(* IEC 61131-3 sources: verifaps-lib/share/PPU.stold (part 19) *)

        Stamp_states_t#StampProcess:
            {* begin(State) *}
            {* begin(onEntry) *}
            Stamp$_transit := FALSE;
            {* end(onEntry) *}
            {* begin(onActive) *}
            Stamp$StampSliderMovedIn := FALSE;
            Stamp$StampPusher := TRUE;
            {* end(onActive) *}
            {* begin(transition) *}
            IF Stamp$StampLowered THEN
                Stamp$_transit := TRUE;
                Stamp$_state := Stamp_states_t#Step1;
            END_IF;
            {* end(transition) *}
            {* begin(onExit) *}
            {* end(onExit) *}
            {* end(State) *}

        Stamp_states_t#StampSliderBack:
            {* begin(State) *}
            {* begin(onEntry) *}
            Stamp$_transit := FALSE;
            {* end(onEntry) *}
            {* begin(onActive) *}
            Stamp$StampSliderMovedIn := TRUE;
            Stamp$StampSliderMovedOut := FALSE;
            {* end(onActive) *}
            {* begin(transition) *}
            IF Stamp$StampSliderSensorMovedIn THEN
                Stamp$_transit := TRUE;
                Stamp$_state := Stamp_states_t#StampProcess;
            END_IF;
            {* end(transition) *}
            {* begin(onExit) *}
            {* end(onExit) *}
            {* end(State) *}

        Stamp_states_t#StampSliderForward:
            {* begin(State) *}
            {* begin(onEntry) *}
            Stamp$_transit := FALSE;
            {* end(onEntry) *}
            {* begin(onActive) *}
            Stamp$StampPusher := FALSE;
            Stamp$StampSliderMovedOut := TRUE;
            IF ((Stamp$StampLowered = FALSE) AND (Stamp$StampUp = TRUE)) THEN
                Stamp$interconnect := FALSE;
            END_IF;
            Stamp$Timer$IN := FALSE;
            Stamp$Timer$PT := USINT#0;
            IF Stamp$Timer$IN THEN
                Stamp$Timer$Q := (Stamp$Timer$ET = USINT#0);
                IF (Stamp$Timer$ET > USINT#0) THEN
                    Stamp$Timer$ET := (Stamp$Timer$ET - USINT#1);
                ELSE
                    Stamp$Timer$ET := USINT#0;
                END_IF;
            ELSE
                Stamp$Timer$Q := FALSE;
                Stamp$Timer$ET := Stamp$Timer$PT;
            END_IF;
            {* end(onActive) *}
            {* begin(transition) *}
            IF Stamp$StampSliderMovedOut THEN
                Stamp$_transit := TRUE;
                Stamp$_state := Stamp_states_t#Step2;
            END_IF;
            {* end(transition) *}
            {* begin(onExit) *}
            {* end(onExit) *}
            {* end(State) *}

        Stamp_states_t#Stamp_Init_1:
            {* begin(State) *}
            {* begin(onEntry) *}
            Stamp$_transit := FALSE;
            {* end(onEntry) *}
            {* begin(onActive) *}
            Stamp$StampSliderMovedIn := TRUE;
            Stamp$StampSliderMovedOut := FALSE;
            {* end(onActive) *}
            {* begin(transition) *}
            IF Stamp$StampSliderSensorMovedIn THEN
                Stamp$_transit := TRUE;
                Stamp$_state := Stamp_states_t#Stamp_Init_2;
            END_IF;
            {* end(transition) *}
            {* begin(onExit) *}
            {* end(onExit) *}
            {* end(State) *}

        Stamp_states_t#Stamp_Init_2:
            {* begin(State) *}
            {* begin(onEntry) *}
            Stamp$_transit := FALSE;
            {* end(onEntry) *}
            {* begin(onActive) *}
            Stamp$StampSliderMovedIn := FALSE;
            Stamp$StampSliderMovedOut := TRUE;
            {* end(onActive) *}
            {* begin(transition) *}
            IF Stamp$StampSliderSensorMovedOut THEN
                Stamp$_transit := TRUE;
                Stamp$_state := Stamp_states_t#Stamp_Init_3;
            END_IF;
            {* end(transition) *}
            {* begin(onExit) *}
            {* end(onExit) *}
            {* end(State) *}

        Stamp_states_t#Stamp_Init_3:
            {* begin(State) *}
            {* begin(onEntry) *}
            Stamp$_transit := FALSE;
            {* end(onEntry) *}
            {* begin(onActive) *}
            Stamp$StampPusher := TRUE;
            {* end(onActive) *}
            {* begin(transition) *}
            IF Stamp$StampLowered THEN
                Stamp$_transit := TRUE;
                Stamp$_state := Stamp_states_t#Stamp_Init_4;
            END_IF;
            {* end(transition) *}
            {* begin(onExit) *}
            {* end(onExit) *}
            {* end(State) *}

        Stamp_states_t#Stamp_Init_4:
            {* begin(State) *}
            {* begin(onEntry) *}
            Stamp$_transit := FALSE;
            {* end(onEntry) *}
            {* begin(onActive) *}
            Stamp$StampPusher := FALSE;
            {* end(onActive) *}
            {* begin(transition) *}
            IF Stamp$StampUp THEN
                Stamp$_transit := TRUE;
                Stamp$_state := Stamp_states_t#Interstep;
            END_IF;
            {* end(transition) *}
            {* begin(onExit) *}
            {* end(onExit) *}
            {* end(State) *}

        Stamp_states_t#Start_Stamp:
            {* begin(State) *}
            {* begin(onEntry) *}
            Stamp$_transit := FALSE;
            {* end(onEntry) *}
            {* begin(onActive) *}
            Stamp$StampSliderMovedOut := FALSE;
            Stamp$StampSliderMovedIn := FALSE;
            Stamp$StampPusher := FALSE;
            Stamp$StampGreenLamp := FALSE;
            Stamp$StampPressure := FALSE;
            Stamp$StartCommandStamp := FALSE;
            IF (Stamp$StampStartButton = TRUE) THEN
                Stamp$interconnectStampStartCommand := TRUE;
            END_IF;
            {* end(onActive) *}
            {* begin(transition) *}
            IF Stamp$interconnectStampStartCommand THEN
                Stamp$_transit := TRUE;
                Stamp$_state := Stamp_states_t#Green_Lamp;
            END_IF;
            {* end(transition) *}
            {* begin(onExit) *}
            {* end(onExit) *}
            {* end(State) *}

        Stamp_states_t#Step0:
            {* begin(State) *}
            {* begin(onEntry) *}
            Stamp$_transit := FALSE;
            {* end(onEntry) *}
            {* begin(onActive) *}
            {* end(onActive) *}
            {* begin(transition) *}
            IF Stamp$CraneUp THEN
                Stamp$_transit := TRUE;
                Stamp$_state := Stamp_states_t#StampSliderBack;
            END_IF;
            {* end(transition) *}
            {* begin(onExit) *}
            {* end(onExit) *}
            {* end(State) *}

        Stamp_states_t#Step1:
            {* begin(State) *}
            {* begin(onEntry) *}
            Stamp$_transit := FALSE;
            {* end(onEntry) *}
            {* begin(onActive) *}
            Stamp$Timer$IN := Stamp$StampLowered;
            Stamp$Timer$PT := USINT#0;
            IF Stamp$Timer$IN THEN
                Stamp$Timer$Q := (Stamp$Timer$ET = USINT#0);
                IF (Stamp$Timer$ET > USINT#0) THEN
                    Stamp$Timer$ET := (Stamp$Timer$ET - USINT#1);
                ELSE
                    Stamp$Timer$ET := USINT#0;
                END_IF;
            ELSE
                Stamp$Timer$Q := FALSE;
                Stamp$Timer$ET := Stamp$Timer$PT;
            END_IF;
            Stamp$interconnect := Stamp$Timer$Q;
            {* end(onActive) *}
            {* begin(transition) *}
            IF Stamp$interconnect THEN
                Stamp$_transit := TRUE;
                Stamp$_state := Stamp_states_t#StampSliderForward;
            END_IF;
            {* end(transition) *}
            {* begin(onExit) *}
            {* end(onExit) *}
            {* end(State) *}

        Stamp_states_t#Step2:
            {* begin(State) *}
            {* begin(onEntry) *}
            Stamp$_transit := FALSE;
            {* end(onEntry) *}
            {* begin(onActive) *}
            {* end(onActive) *}
            {* begin(transition) *}
            IF (((Stamp$AnalogCranePosition > INT#16160) AND (Stamp$AnalogCranePosition < INT#16260)) AND NOT Stamp$StampSliderFilled) THEN
                Stamp$_transit := TRUE;
                Stamp$_state := Stamp_states_t#Interstep;
            END_IF;
            {* end(transition) *}
            {* begin(onExit) *}
            {* end(onExit) *}
            {* end(State) *}

            END_CASE;
    CASE Conveyor$_state OF
        Conveyor_states_t#Conveyor_Init:
            {* begin(State) *}
            {* begin(onEntry) *}
            Conveyor$_transit := FALSE;
            {* end(onEntry) *}
            {* begin(onActive) *}
            Conveyor$SorterConveyorTowardsStacker := TRUE;
            Conveyor$SorterConveyorTowardsCrane := FALSE;
            Conveyor$Timer_Conveyor_Test$IN := TRUE;
            Conveyor$Timer_Conveyor_Test$PT := Conveyor$Duration_Conveyor_Test;
            IF Conveyor$Timer_Conveyor_Test$IN THEN
                Conveyor$Timer_Conveyor_Test$Q := (Conveyor$Timer_Conveyor_Test$ET = USINT#0);
                IF (Conveyor$Timer_Conveyor_Test$ET > USINT#0) THEN
                    Conveyor$Timer_Conveyor_Test$ET := (Conveyor$Timer_Conveyor_Test$ET - USINT#1);
                ELSE
                    Conveyor$Timer_Conveyor_Test$ET := USINT#0;
                END_IF;
            ELSE
                Conveyor$Timer_Conveyor_Test$Q := FALSE;
                Conveyor$Timer_Conveyor_Test$ET := Conveyor$Timer_Conveyor_Test$PT;
            END_IF;
            Conveyor$interconnect_Conveyor_Test := Conveyor$Timer_Conveyor_Test$Q;
            {* end(onActive) *}
            {* begin(transition) *}
            IF Conveyor$interconnect_Conveyor_Test THEN
                Conveyor$_transit := TRUE;
                Conveyor$_state := Conveyor_states_t#Conveyor_init_2;
            END_IF;
            {* end(transition) *}
            {* begin(onExit) *}
            {* end(onExit) *}
            {* end(State) *}

        Conveyor_states_t#Conveyor_Stop_Empty_Magazin:
            {* begin(State) *}
            {* begin(onEntry) *}
            Conveyor$_transit := FALSE;
            {* end(onEntry) *}
            {* begin(onActive) *}
            Conveyor$SorterConveyorTowardsStacker := FALSE;
            Conveyor$SorterConveyorTowardsCrane := FALSE;
            Conveyor$interconnectConveyorStartCommand := FALSE;
            {* end(onActive) *}
            {* begin(transition) *}
            IF TRUE THEN
                Conveyor$_transit := TRUE;
                Conveyor$_state := Conveyor_states_t#Interstep;
            END_IF;
            {* end(transition) *}
            {* begin(onExit) *}
            {* end(onExit) *}
            {* end(State) *}

        Conveyor_states_t#Conveyor_Towards_Stacker:
            {* begin(State) *}
            {* begin(onEntry) *}
            Conveyor$_transit := FALSE;
            {* end(onEntry) *}
            {* begin(onActive) *}
            Conveyor$SorterConveyorTowardsStacker := TRUE;
            Conveyor$SorterConveyorTowardsCrane := FALSE;
            {* end(onActive) *}
            {* begin(transition) *}
            IF TRUE THEN
                Conveyor$_transit := TRUE;
                Conveyor$_state := Conveyor_states_t#Runtime_Conveyor;
            END_IF;
            {* end(transition) *}
            {* begin(onExit) *}
            {* end(onExit) *}
            {* end(State) *}

        Conveyor_states_t#Conveyor_init_2:
            {* begin(State) *}
            {* begin(onEntry) *}
            Conveyor$_transit := FALSE;
            {* end(onEntry) *}
            {* begin(onActive) *}
            Conveyor$SorterConveyorTowardsStacker := FALSE;
            Conveyor$SorterConveyorTowardsCrane := FALSE;
            Conveyor$interconnect_Conveyor_Test := FALSE;
            Conveyor$Timer_Conveyor_Test$IN := FALSE;
            Conveyor$Timer_Conveyor_Test$PT := USINT#0;
            IF Conveyor$Timer_Conveyor_Test$IN THEN
                Conveyor$Timer_Conveyor_Test$Q := (Conveyor$Timer_Conveyor_Test$ET = USINT#0);
                IF (Conveyor$Timer_Conveyor_Test$ET > USINT#0) THEN
                    Conveyor$Timer_Conveyor_Test$ET := (Conveyor$Timer_Conveyor_Test$ET - USINT#1);
                ELSE
                    Conveyor$Timer_Conveyor_Test$ET := USINT#0;
                END_IF;
            ELSE
                Conveyor$Timer_Conveyor_Test$Q := FALSE;
                Conveyor$Timer_Conveyor_Test$ET := Conveyor$Timer_Conveyor_Test$PT;
            END_IF;
            {* end(onActive) *}
            {* begin(transition) *}
            IF TRUE THEN
                Conveyor$_transit := TRUE;
                Conveyor$_state := Conveyor_states_t#Interstep;
            END_IF;
            {* end(transition) *}
            {* begin(onExit) *}
            {* end(onExit) *}
            {* end(State) *}

        Conveyor_states_t#Conveyor_pause:
            {* begin(State) *}
            {* begin(onEntry) *}
            Conveyor$_transit := FALSE;
            {* end(onEntry) *}
            {* begin(onActive) *}
            Conveyor$SorterConveyorTowardsStacker := FALSE;
            Conveyor$SorterConveyorTowardsCrane := FALSE;
            Conveyor$interconnect_Conveyor_Runtime := FALSE;
            Conveyor$Timer_Conveyor_Runtime$IN := FALSE;
            Conveyor$Timer_Conveyor_Runtime$PT := USINT#0;
            IF Conveyor$Timer_Conveyor_Runtime$IN THEN
                Conveyor$Timer_Conveyor_Runtime$Q := (Conveyor$Timer_Conveyor_Runtime$ET = USINT#0);
                IF (Conveyor$Timer_Conveyor_Runtime$ET > USINT#0) THEN
                    Conveyor$Timer_Conveyor_Runtime$ET := (Conveyor$Timer_Conveyor_Runtime$ET - USINT#1);
                ELSE
                    Conveyor$Timer_Conveyor_Runtime$ET := USINT#0;
                END_IF;
            ELSE
                Conveyor$Timer_Conveyor_Runtime$Q := FALSE;
                Conveyor$Timer_Conveyor_Runtime$ET := Conveyor$Timer_Conveyor_Runtime$PT;
            END_IF;
            {* end(onActive) *}
            {* begin(transition) *}
            IF TRUE THEN
                Conveyor$_transit := TRUE;
                Conveyor$_state := Conveyor_states_t#Interstep;
            END_IF;
            {* end(transition) *}
            {* begin(onExit) *}
            {* end(onExit) *}
            {* end(State) *}

        Conveyor_states_t#Green_Lamp:
            {* begin(State) *}
            {* begin(onEntry) *}
            Conveyor$_transit := FALSE;
            {* end(onEntry) *}
            {* begin(onActive) *}
            Conveyor$SorterGreenLampConveyor := TRUE;
            Conveyor$interconnectConveyorStartCommand := FALSE;
            {* end(onActive) *}
            {* begin(transition) *}
            IF TRUE THEN
                Conveyor$_transit := TRUE;
                Conveyor$_state := Conveyor_states_t#Conveyor_Init;
            END_IF;
            {* end(transition) *}
            {* begin(onExit) *}
            {* end(onExit) *}
            {* end(State) *}

        Conveyor_states_t#Init:
            {* begin(State) *}
            {* begin(onEntry) *}
            Conveyor$_transit := FALSE;
            {* end(onEntry) *}
            {* begin(onActive) *}
            {* end(onActive) *}
            {* begin(transition) *}
            IF TRUE THEN
                Conveyor$_transit := TRUE;
                Conveyor$_state := Conveyor_states_t#Start_Conveyor;
            END_IF;
            {* end(transition) *}
            {* begin(onExit) *}
            {* end(onExit) *}
            {* end(State) *}

        Conveyor_states_t#Interstep:
            {* begin(State) *}
            {* begin(onEntry) *}
            Conveyor$_transit := FALSE;
            {* end(onEntry) *}
            {* begin(onActive) *}
            Conveyor$StartCommandConveyor := TRUE;
            {* end(onActive) *}
            {* begin(transition) *}
            IF Conveyor$StartVar THEN
                Conveyor$_transit := TRUE;
                Conveyor$_state := Conveyor_states_t#Step0;
            END_IF;
            {* end(transition) *}
            {* begin(onExit) *}
            {* end(onExit) *}
            {* end(State) *}

        Conveyor_states_t#Runtime_Conveyor:
            {* begin(State) *}
            {* begin(onEntry) *}
            Conveyor$_transit := FALSE;
            {* end(onEntry) *}
            {* begin(onActive) *}
            Conveyor$Timer_Conveyor_Runtime$IN := TRUE;
            Conveyor$Timer_Conveyor_Runtime$PT := Conveyor$Duration_Conveyor_Runtime;
            IF Conveyor$Timer_Conveyor_Runtime$IN THEN
                Conveyor$Timer_Conveyor_Runtime$Q := (Conveyor$Timer_Conveyor_Runtime$ET = USINT#0);
                IF (Conveyor$Timer_Conveyor_Runtime$ET > USINT#0) THEN
                    Conveyor$Timer_Conveyor_Runtime$ET := (Conveyor$Timer_Conveyor_Runtime$ET - USINT#1);
                ELSE
                    Conveyor$Timer_Conveyor_Runtime$ET := USINT#0;
                END_IF;
            ELSE
                Conveyor$Timer_Conveyor_Runtime$Q := FALSE;
                Conveyor$Timer_Conveyor_Runtime$ET := Conveyor$Timer_Conveyor_Runtime$PT;
            END_IF;
            Conveyor$interconnect_Conveyor_Runtime := Conveyor$Timer_Conveyor_Runtime$Q;
            {* end(onActive) *}
            {* begin(transition) *}
            IF Conveyor$interconnect_Conveyor_Runtime THEN
                Conveyor$_transit := TRUE;
                Conveyor$_state := Conveyor_states_t#Conveyor_pause;
            END_IF;
            {* end(transition) *}
            {* begin(onExit) *}
            {* end(onExit) *}
            {* end(State) *}

        Conveyor_states_t#Start_Conveyor:
            {* begin(State) *}
            {* begin(onEntry) *}
            Conveyor$_transit := FALSE;
            {* end(onEntry) *}
            {* begin(onActive) *}
            Conveyor$interconnectConveyorTerminationCommand := FALSE;
            Conveyor$SorterConveyorTowardsStacker := FALSE;
            Conveyor$SorterConveyorTowardsCrane := FALSE;
            Conveyor$SorterGreenLampConveyor := FALSE;
            Conveyor$interconnect_Conveyor_Runtime := FALSE;
            Conveyor$interconnect_Conveyor_Test := FALSE;
            Conveyor$Timer_Conveyor_Test$IN := FALSE;
            Conveyor$Timer_Conveyor_Test$PT := USINT#0;
            IF Conveyor$Timer_Conveyor_Test$IN THEN
                Conveyor$Timer_Conveyor_Test$Q := (Conveyor$Timer_Conveyor_Test$ET = USINT#0);
                IF (Conveyor$Timer_Conveyor_Test$ET > USINT#0) THEN
                    Conveyor$Timer_Conveyor_Test$ET := (Conveyor$Timer_Conveyor_Test$ET - USINT#1);
                ELSE
                    Conveyor$Timer_Conveyor_Test$ET := USINT#0;
                END_IF;
            ELSE
                Conveyor$Timer_Conveyor_Test$Q := FALSE;
                Conveyor$Timer_Conveyor_Test$ET := Conveyor$Timer_Conveyor_Test$PT;
            END_IF;
            Conveyor$Timer_Conveyor_Runtime$IN := FALSE;
            Conveyor$Timer_Conveyor_Runtime$PT := USINT#0;
            IF Conveyor$Timer_Conveyor_Runtime$IN THEN
                Conveyor$Timer_Conveyor_Runtime$Q := (Conveyor$Timer_Conveyor_Runtime$ET = USINT#0);
                IF (Conveyor$Timer_Conveyor_Runtime$ET > USINT#0) THEN
                    Conveyor$Timer_Conveyor_Runtime$ET := (Conveyor$Timer_Conveyor_Runtime$ET - USINT#1);
                ELSE
                    Conveyor$Timer_Conveyor_Runtime$ET := USINT#0;
                END_IF;
            ELSE
                Conveyor$Timer_Conveyor_Runtime$Q := FALSE;
                Conveyor$Timer_Conveyor_Runtime$ET := Conveyor$Timer_Conveyor_Runtime$PT;
            END_IF;
            Conveyor$StartVar := FALSE;
            Conveyor$StartCommandConveyor := FALSE;
            IF (Conveyor$SorterStartButton = TRUE) THEN
                Conveyor$interconnectConveyorStartCommand := TRUE;
            END_IF;
            {* end(onActive) *}
            {* begin(transition) *}
            IF Conveyor$interconnectConveyorStartCommand THEN
                Conveyor$_transit := TRUE;
                Conveyor$_state := Conveyor_states_t#Green_Lamp;
            END_IF;
            {* end(transition) *}
            {* begin(onExit) *}
            {* end(onExit) *}
            {* end(State) *}

        Conveyor_states_t#Step0:
            {* begin(State) *}
            {* begin(onEntry) *}
            Conveyor$_transit := FALSE;
            {* end(onEntry) *}
            {* begin(onActive) *}
            {* end(onActive) *}
            {* begin(transition) *}
            IF Conveyor$SorterLightbarrierCraneInterface THEN
                Conveyor$_transit := TRUE;
                Conveyor$_state := Conveyor_states_t#Conveyor_Towards_Stacker;
            ELSEIF NOT Conveyor$SorterLightbarrierCraneInterface THEN
                Conveyor$_transit := TRUE;
                Conveyor$_state := Conveyor_states_t#Conveyor_Stop_Empty_Magazin;
            END_IF;
            {* end(transition) *}
            {* begin(onExit) *}
            {* end(onExit) *}
            {* end(State) *}

            END_CASE;
    CASE Pusher$_state OF
        Pusher_states_t#Check_For_Black:
            {* begin(State) *}
            {* begin(onEntry) *}
            Pusher$_transit := FALSE;
            {* end(onEntry) *}
            {* begin(onActive) *}
            {* end(onActive) *}
            {* begin(transition) *}
            IF ((Pusher$Slide2_black = INT#1) AND (Pusher$Priority_Var_Black = INT#2)) THEN
                Pusher$_transit := TRUE;
                Pusher$_state := Pusher_states_t#Second_Slide_black_workpieces;
            ELSEIF ((Pusher$Slide3_black = INT#1) AND (Pusher$Priority_Var_Black = INT#3)) THEN
                Pusher$_transit := TRUE;
                Pusher$_state := Pusher_states_t#Third_Slide_black_workpieces;
            ELSEIF ((Pusher$Slide1_black = INT#1) AND (Pusher$Priority_Var_Black = INT#1)) THEN
                Pusher$_transit := TRUE;
                Pusher$_state := Pusher_states_t#First_Slide_black_workpieces;
            END_IF;
            {* end(transition) *}
            {* begin(onExit) *}
            {* end(onExit) *}
            {* end(State) *}

        Pusher_states_t#Check_For_Metal:
            {* begin(State) *}
            {* begin(onEntry) *}
            Pusher$_transit := FALSE;
            {* end(onEntry) *}
            {* begin(onActive) *}
            {* end(onActive) *}
            {* begin(transition) *}
            IF ((Pusher$Slide3_metal = INT#1) AND (Pusher$Priority_Var_Metal = INT#3)) THEN
                Pusher$_transit := TRUE;
                Pusher$_state := Pusher_states_t#Third_Slide_metal_workpieces;
            ELSEIF ((Pusher$Slide2_metal = INT#1) AND (Pusher$Priority_Var_Metal = INT#2)) THEN
                Pusher$_transit := TRUE;
                Pusher$_state := Pusher_states_t#Second_Slide_metal_workpieces;
            ELSEIF ((Pusher$Slide1_metal = INT#1) AND (Pusher$Priority_Var_Metal = INT#1)) THEN
                Pusher$_transit := TRUE;
                Pusher$_state := Pusher_states_t#First_Slide_metal_workpieces;
            END_IF;
            {* end(transition) *}
            {* begin(onExit) *}
            {* end(onExit) *}
            {* end(State) *}

        Pusher_states_t#Check_For_White:
            {* begin(State) *}
            {* begin(onEntry) *}
            Pusher$_transit := FALSE;
            {* end(onEntry) *}
            {* begin(onActive) *}
            {* end(onActive) *}
            {* begin(transition) *}
            IF ((Pusher$Slide1_white = INT#1) AND (Pusher$Priority_Var_White = INT#1)) THEN
                Pusher$_transit := TRUE;
                Pusher$_state := Pusher_states_t#First_Slide_white_workpieces;
            ELSEIF ((Pusher$Slide3_white = INT#1) AND (Pusher$Priority_Var_White = INT#3)) THEN
                Pusher$_transit := TRUE;
                Pusher$_state := Pusher_states_t#Third_Slide_white_workpieces;
            ELSEIF ((Pusher$Slide2_white = INT#1) AND (Pusher$Priority_Var_White = INT#2)) THEN
                Pusher$_transit := TRUE;
                Pusher$_state := Pusher_states_t#Second_Slide_white_workpieces;
            END_IF;
            {* end(transition) *}
            {* begin(onExit) *}
            {* end(onExit) *}
            {* end(State) *}

        Pusher_states_t#First_Slide_Timer_Black:
            {* begin(State) *}
            {* begin(onEntry) *}
            Pusher$_transit := FALSE;
            {* end(onEntry) *}
            {* begin(onActive) *}
            IF (Pusher$SorterLightnesssensorCraneInterfaceInverse = TRUE) THEN
                Pusher$Timer_Slide1_Black$IN := Pusher$SorterLightnesssensorCraneInterfaceInverse;
                Pusher$Timer_Slide1_Black$PT := Pusher$Duration_Slide1_Black;
                IF Pusher$Timer_Slide1_Black$IN THEN
                    Pusher$Timer_Slide1_Black$Q := (Pusher$Timer_Slide1_Black$ET = USINT#0);
                    IF (Pusher$Timer_Slide1_Black$ET > USINT#0) THEN
                        Pusher$Timer_Slide1_Black$ET := (Pusher$Timer_Slide1_Black$ET - USINT#1);
                    ELSE
                        Pusher$Timer_Slide1_Black$ET := USINT#0;
                    END_IF;
                ELSE
                    Pusher$Timer_Slide1_Black$Q := FALSE;
                    Pusher$Timer_Slide1_Black$ET := Pusher$Timer_Slide1_Black$PT;
                END_IF;
                Pusher$interconnect_Slide1_Black := Pusher$Timer_Slide1_Black$Q;
            END_IF;
            {* end(onActive) *}
            {* begin(transition) *}
            IF Pusher$interconnect_Slide1_Black THEN
                Pusher$_transit := TRUE;
                Pusher$_state := Pusher_states_t#PusherY1_Move_Out_Black;
            END_IF;
            {* end(transition) *}
            {* begin(onExit) *}
            {* end(onExit) *}
            {* end(State) *}

        Pusher_states_t#First_Slide_Timer_Metal:
            {* begin(State) *}
            {* begin(onEntry) *}
            Pusher$_transit := FALSE;
            {* end(onEntry) *}
            {* begin(onActive) *}
            Pusher$Timer_Slide1_Metal$IN := TRUE;
            Pusher$Timer_Slide1_Metal$PT := Pusher$Duration_Slide1_Metal;
            IF Pusher$Timer_Slide1_Metal$IN THEN
                Pusher$Timer_Slide1_Metal$Q := (Pusher$Timer_Slide1_Metal$ET = USINT#0);
                IF (Pusher$Timer_Slide1_Metal$ET > USINT#0) THEN
                    Pusher$Timer_Slide1_Metal$ET := (Pusher$Timer_Slide1_Metal$ET - USINT#1);
                ELSE
                    Pusher$Timer_Slide1_Metal$ET := USINT#0;
                END_IF;
            ELSE
                Pusher$Timer_Slide1_Metal$Q := FALSE;
                Pusher$Timer_Slide1_Metal$ET := Pusher$Timer_Slide1_Metal$PT;
            END_IF;
            Pusher$interconnect_Slide1_Metal := Pusher$Timer_Slide1_Metal$Q;
            {* end(onActive) *}
            {* begin(transition) *}
            IF Pusher$interconnect_Slide1_Metal THEN
                Pusher$_transit := TRUE;
                Pusher$_state := Pusher_states_t#PusherY1_Move_Out_Metal;
            END_IF;
            {* end(transition) *}
            {* begin(onExit) *}
            {* end(onExit) *}
            {* end(State) *}

        Pusher_states_t#First_Slide_Timer_White:
            {* begin(State) *}
            {* begin(onEntry) *}
            Pusher$_transit := FALSE;
            {* end(onEntry) *}
            {* begin(onActive) *}
            Pusher$Timer_Slide1_White$IN := TRUE;
            Pusher$Timer_Slide1_White$PT := Pusher$Duration_Slide1_White;
            IF Pusher$Timer_Slide1_White$IN THEN
                Pusher$Timer_Slide1_White$Q := (Pusher$Timer_Slide1_White$ET = USINT#0);
                IF (Pusher$Timer_Slide1_White$ET > USINT#0) THEN
                    Pusher$Timer_Slide1_White$ET := (Pusher$Timer_Slide1_White$ET - USINT#1);
                ELSE
                    Pusher$Timer_Slide1_White$ET := USINT#0;
                END_IF;
            ELSE
                Pusher$Timer_Slide1_White$Q := FALSE;
                Pusher$Timer_Slide1_White$ET := Pusher$Timer_Slide1_White$PT;
            END_IF;
            Pusher$interconnect_Slide1_White := Pusher$Timer_Slide1_White$Q;
            {* end(onActive) *}
            {* begin(transition) *}
            IF Pusher$interconnect_Slide1_White THEN
                Pusher$_transit := TRUE;
                Pusher$_state := Pusher_states_t#PusherY1_Move_Out_White;
            END_IF;
            {* end(transition) *}
            {* begin(onExit) *}
            {* end(onExit) *}
            {* end(State) *}

        Pusher_states_t#First_Slide_black_workpieces:
            {* begin(State) *}
            {* begin(onEntry) *}
            Pusher$_transit := FALSE;
            {* end(onEntry) *}
            {* begin(onActive) *}
            {* end(onActive) *}
            {* begin(transition) *}
            IF TRUE THEN
                Pusher$_transit := TRUE;
                Pusher$_state := Pusher_states_t#First_Slide_Timer_Black;
            END_IF;
            {* end(transition) *}
            {* begin(onExit) *}
            {* end(onExit) *}
            {* end(State) *}

        Pusher_states_t#First_Slide_metal_workpieces:
            {* begin(State) *}
            {* begin(onEntry) *}
            Pusher$_transit := FALSE;
            {* end(onEntry) *}
            {* begin(onActive) *}
            {* end(onActive) *}
            {* begin(transition) *}
            IF TRUE THEN
                Pusher$_transit := TRUE;
                Pusher$_state := Pusher_states_t#First_Slide_Timer_Metal;
            END_IF;
            {* end(transition) *}
            {* begin(onExit) *}
            {* end(onExit) *}
            {* end(State) *}

        Pusher_states_t#First_Slide_white_workpieces:
            {* begin(State) *}
            {* begin(onEntry) *}
            Pusher$_transit := FALSE;
            {* end(onEntry) *}
            {* begin(onActive) *}
            {* end(onActive) *}
            {* begin(transition) *}
            IF TRUE THEN
                Pusher$_transit := TRUE;
                Pusher$_state := Pusher_states_t#First_Slide_Timer_White;
            END_IF;
            {* end(transition) *}
            {* begin(onExit) *}
            {* end(onExit) *}
            {* end(State) *}

        Pusher_states_t#Init:
            {* begin(State) *}
            {* begin(onEntry) *}
            Pusher$_transit := FALSE;
            {* end(onEntry) *}
            {* begin(onActive) *}
            {* end(onActive) *}
            {* begin(transition) *}
            IF Pusher$StartVar THEN
                Pusher$_transit := TRUE;
                Pusher$_state := Pusher_states_t#Interstep;
            END_IF;
            {* end(transition) *}
            {* begin(onExit) *}
            {* end(onExit) *}
            {* end(State) *}

        Pusher_states_t#Interstep:
            {* begin(State) *}
            {* begin(onEntry) *}
            Pusher$_transit := FALSE;
            {* end(onEntry) *}
            {* begin(onActive) *}
            Pusher$PusherY1 := FALSE;
            Pusher$PusherY2 := FALSE;
            Pusher$interconnect2 := FALSE;
            Pusher$interconnect3 := FALSE;
            Pusher$StartVar := FALSE;
            Pusher$interconnect_Slide1_Black := FALSE;
            Pusher$interconnect_Slide2_Black := FALSE;
            Pusher$interconnect_Slide1_White := FALSE;
            Pusher$interconnect_Slide2_White := FALSE;
            Pusher$interconnect_Slide1_Metal := FALSE;
            Pusher$interconnect_Slide2_Metal := FALSE;
            {* end(onActive) *}
            {* begin(transition) *}
            IF TRUE THEN
                Pusher$_transit := TRUE;
                Pusher$_state := Pusher_states_t#Interstep_2;
            END_IF;
            {* end(transition) *}
            {* begin(onExit) *}
            {* end(onExit) *}
            {* end(State) *}

        Pusher_states_t#Interstep_2:
            {* begin(State) *}
            {* begin(onEntry) *}
            Pusher$_transit := FALSE;
            {* end(onEntry) *}
            {* begin(onActive) *}
            {* end(onActive) *}
            {* begin(transition) *}
            IF ((Pusher$SorterLightnessSensorPusher1 AND Pusher$SorterCapacitiveSensorPusher1) AND (Pusher$Priority_Var_Metal > INT#0)) THEN
                Pusher$_transit := TRUE;
                Pusher$_state := Pusher_states_t#Check_For_Metal;
            ELSEIF ((NOT Pusher$SorterLightnesssensorCraneInterfaceInverse AND Pusher$SorterLightbarrierCraneInterface) AND (Pusher$Priority_Var_Black > INT#0)) THEN
                Pusher$_transit := TRUE;
                Pusher$_state := Pusher_states_t#Check_For_Black;
            ELSEIF ((Pusher$SorterLightnessSensorPusher1 AND NOT Pusher$SorterCapacitiveSensorPusher1) AND (Pusher$Priority_Var_White > INT#0)) THEN
                Pusher$_transit := TRUE;
                Pusher$_state := Pusher_states_t#Check_For_White;
            END_IF;
            {* end(transition) *}
            {* begin(onExit) *}
            {* end(onExit) *}
            {* end(State) *}

        Pusher_states_t#PusherY1_Move_In_Black:
            {* begin(State) *}
            {* begin(onEntry) *}
            Pusher$_transit := FALSE;
            {* end(onEntry) *}
            {* begin(onActive) *}
            IF ((Pusher$SorterPusher1MovedOut = TRUE) AND (Pusher$SorterPusher1MovedIn = FALSE)) THEN
                Pusher$PusherY1 := FALSE;
            END_IF;
            {* end(onActive) *}
            {* begin(transition) *}
            IF Pusher$SorterPusher1MovedIn THEN
                Pusher$_transit := TRUE;
                Pusher$_state := Pusher_states_t#Reset_interconnect_Slide1_Black;
            END_IF;
            {* end(transition) *}
            {* begin(onExit) *}
            {* end(onExit) *}
            {* end(State) *}

        Pusher_states_t#PusherY1_Move_In_Metal:
            {* begin(State) *}
            {* begin(onEntry) *}
            Pusher$_transit := FALSE;
            {* end(onEntry) *}
            {* begin(onActive) *}
            IF ((Pusher$SorterPusher1MovedOut = TRUE) AND (Pusher$SorterPusher1MovedIn = FALSE)) THEN
                Pusher$PusherY1 := FALSE;
            END_IF;
            {* end(onActive) *}
            {* begin(transition) *}
            IF Pusher$SorterPusher1MovedIn THEN
                Pusher$_transit := TRUE;
                Pusher$_state := Pusher_states_t#Reset_interconnect_Slide1_Metal;
            END_IF;
            {* end(transition) *}
            {* begin(onExit) *}
            {* end(onExit) *}
            {* end(State) *}

        Pusher_states_t#PusherY1_Move_In_White:
            {* begin(State) *}
            {* begin(onEntry) *}
            Pusher$_transit := FALSE;
            {* end(onEntry) *}
            {* begin(onActive) *}
            IF ((Pusher$SorterPusher1MovedOut = TRUE) AND (Pusher$SorterPusher1MovedIn = FALSE)) THEN
                Pusher$PusherY1 := FALSE;
            END_IF;
            {* end(onActive) *}
            {* begin(transition) *}
            IF Pusher$SorterPusher1MovedIn THEN
                Pusher$_transit := TRUE;
                Pusher$_state := Pusher_states_t#Reset_interconnect_Slide1_White;
            END_IF;
            {* end(transition) *}
            {* begin(onExit) *}
            {* end(onExit) *}
            {* end(State) *}

        Pusher_states_t#PusherY1_Move_Out_Black:
            {* begin(State) *}
            {* begin(onEntry) *}
            Pusher$_transit := FALSE;
            {* end(onEntry) *}
            {* begin(onActive) *}
            IF ((Pusher$SorterPusher1MovedOut = FALSE) AND (Pusher$SorterPusher1MovedIn = TRUE)) THEN
                Pusher$PusherY1 := TRUE;
            END_IF;
            {* end(onActive) *}
            {* begin(transition) *}
            IF Pusher$SorterPusher1MovedOut THEN
                Pusher$_transit := TRUE;
                Pusher$_state := Pusher_states_t#Wait_Y1_Black;
            END_IF;
            {* end(transition) *}
            {* begin(onExit) *}
            {* end(onExit) *}
            {* end(State) *}

        Pusher_states_t#PusherY1_Move_Out_Metal:
            {* begin(State) *}
            {* begin(onEntry) *}
            Pusher$_transit := FALSE;
            {* end(onEntry) *}
            {* begin(onActive) *}
            IF ((Pusher$SorterPusher1MovedOut = FALSE) AND (Pusher$SorterPusher1MovedIn = TRUE)) THEN
                Pusher$PusherY1 := TRUE;
            END_IF;
            {* end(onActive) *}
            {* begin(transition) *}
            IF Pusher$SorterPusher1MovedOut THEN
                Pusher$_transit := TRUE;
                Pusher$_state := Pusher_states_t#Wait_Y1_Metal;
            END_IF;
            {* end(transition) *}
            {* begin(onExit) *}
            {* end(onExit) *}
            {* end(State) *}

        Pusher_states_t#PusherY1_Move_Out_White:
            {* begin(State) *}
            {* begin(onEntry) *}
            Pusher$_transit := FALSE;
            {* end(onEntry) *}
            {* begin(onActive) *}
            IF ((Pusher$SorterPusher1MovedOut = FALSE) AND (Pusher$SorterPusher1MovedIn = TRUE)) THEN
                Pusher$PusherY1 := TRUE;
            END_IF;
            {* end(onActive) *}
            {* begin(transition) *}
            IF Pusher$SorterPusher1MovedOut THEN
                Pusher$_transit := TRUE;
                Pusher$_state := Pusher_states_t#Wait_Y1_White;
            END_IF;
            {* end(transition) *}
            {* begin(onExit) *}
            {* end(onExit) *}
            {* end(State) *}

        Pusher_states_t#PusherY2_Move_In_Black:
            {* begin(State) *}
            {* begin(onEntry) *}
            Pusher$_transit := FALSE;
            {* end(onEntry) *}
            {* begin(onActive) *}
            IF ((Pusher$SorterPusher2MovedOut = TRUE) AND (Pusher$SorterPusher2MovedIn = FALSE)) THEN
                Pusher$PusherY2 := FALSE;
            END_IF;
            {* end(onActive) *}
            {* begin(transition) *}
            IF Pusher$SorterPusher2MovedIn THEN
                Pusher$_transit := TRUE;
                Pusher$_state := Pusher_states_t#Reset_interconnect_Slide2_Black;
            END_IF;
            {* end(transition) *}
            {* begin(onExit) *}
            {* end(onExit) *}
            {* end(State) *}

        Pusher_states_t#PusherY2_Move_In_Metal:
            {* begin(State) *}
            {* begin(onEntry) *}
            Pusher$_transit := FALSE;
            {* end(onEntry) *}
            {* begin(onActive) *}
            IF ((Pusher$SorterPusher2MovedOut = TRUE) AND (Pusher$SorterPusher2MovedIn = FALSE)) THEN
                Pusher$PusherY2 := FALSE;
            END_IF;
            {* end(onActive) *}
            {* begin(transition) *}
            IF Pusher$SorterPusher2MovedIn THEN
                Pusher$_transit := TRUE;
                Pusher$_state := Pusher_states_t#Reset_interconnect_Slide2_Metal;
            END_IF;
            {* end(transition) *}
            {* begin(onExit) *}
            {* end(onExit) *}
            {* end(State) *}

        Pusher_states_t#PusherY2_Move_In_White:
            {* begin(State) *}
            {* begin(onEntry) *}
            Pusher$_transit := FALSE;
            {* end(onEntry) *}
            {* begin(onActive) *}
            IF ((Pusher$SorterPusher2MovedOut = TRUE) AND (Pusher$SorterPusher2MovedIn = FALSE)) THEN
                Pusher$PusherY2 := FALSE;
            END_IF;
            {* end(onActive) *}
            {* begin(transition) *}
            IF Pusher$SorterPusher2MovedIn THEN
                Pusher$_transit := TRUE;
                Pusher$_state := Pusher_states_t#Reset_interconnect_Slide2_White;
            END_IF;
            {* end(transition) *}
            {* begin(onExit) *}
            {* end(onExit) *}
            {* end(State) *}

        Pusher_states_t#PusherY2_Move_Out_Black:
            {* begin(State) *}
            {* begin(onEntry) *}
            Pusher$_transit := FALSE;
            {* end(onEntry) *}
            {* begin(onActive) *}
            IF ((Pusher$SorterPusher2MovedOut = FALSE) AND (Pusher$SorterPusher2MovedIn = TRUE)) THEN
                Pusher$PusherY2 := TRUE;
            END_IF;
            {* end(onActive) *}
            {* begin(transition) *}
            IF Pusher$SorterPusher2MovedOut THEN
                Pusher$_transit := TRUE;
                Pusher$_state := Pusher_states_t#Wait_Y2_Black;
            END_IF;
            {* end(transition) *}
            {* begin(onExit) *}
            {* end(onExit) *}
            {* end(State) *}

        Pusher_states_t#PusherY2_Move_Out_Metal:
            {* begin(State) *}
            {* begin(onEntry) *}
            Pusher$_transit := FALSE;
            {* end(onEntry) *}
            {* begin(onActive) *}
            IF ((Pusher$SorterPusher2MovedOut = FALSE) AND (Pusher$SorterPusher2MovedIn = TRUE)) THEN
                Pusher$PusherY2 := TRUE;
            END_IF;
            {* end(onActive) *}
            {* begin(transition) *}
            IF Pusher$SorterPusher2MovedOut THEN
                Pusher$_transit := TRUE;
                Pusher$_state := Pusher_states_t#Wait_Y2_Metal;
            END_IF;
            {* end(transition) *}
            {* begin(onExit) *}
            {* end(onExit) *}
            {* end(State) *}

        Pusher_states_t#PusherY2_Move_Out_White:
            {* begin(State) *}
            {* begin(onEntry) *}
            Pusher$_transit := FALSE;
            {* end(onEntry) *}
            {* begin(onActive) *}
            IF ((Pusher$SorterPusher2MovedOut = FALSE) AND (Pusher$SorterPusher2MovedIn = TRUE)) THEN
                Pusher$PusherY2 := TRUE;
            END_IF;
            {* end(onActive) *}
            {* begin(transition) *}
            IF Pusher$SorterPusher2MovedOut THEN
                Pusher$_transit := TRUE;
                Pusher$_state := Pusher_states_t#Wait_Y2_White;
            END_IF;
            {* end(transition) *}
            {* begin(onExit) *}
            {* end(onExit) *}
            {* end(State) *}

        Pusher_states_t#Reset_interconnect3:
            {* begin(State) *}
            {* begin(onEntry) *}
            Pusher$_transit := FALSE;
            {* end(onEntry) *}
            {* begin(onActive) *}
            Pusher$interconnect2 := FALSE;
            Pusher$Timer2$IN := FALSE;
            Pusher$Timer2$PT := USINT#0;
            IF Pusher$Timer2$IN THEN
                Pusher$Timer2$Q := (Pusher$Timer2$ET = USINT#0);
                IF (Pusher$Timer2$ET > USINT#0) THEN
                    Pusher$Timer2$ET := (Pusher$Timer2$ET - USINT#1);
                ELSE
                    Pusher$Timer2$ET := USINT#0;
                END_IF;
            ELSE
                Pusher$Timer2$Q := FALSE;
                Pusher$Timer2$ET := Pusher$Timer2$PT;
            END_IF;
            Pusher$Slide3_black := (Pusher$Slide3_black - INT#1);
            Pusher$Priority_Var_Black := (Pusher$Priority_Var_Black - INT#1);
            {* end(onActive) *}
            {* begin(transition) *}
            IF TRUE THEN
                Pusher$_transit := TRUE;
                Pusher$_state := Pusher_states_t#Interstep_2;
            END_IF;
            {* end(transition) *}
            {* begin(onExit) *}
            {* end(onExit) *}
            {* end(State) *}

        Pusher_states_t#Reset_interconnect_Slide1_Black:
            {* begin(State) *}
            {* begin(onEntry) *}
            Pusher$_transit := FALSE;
            {* end(onEntry) *}
            {* begin(onActive) *}
            Pusher$interconnect3 := FALSE;
            Pusher$Timer3$IN := FALSE;
            Pusher$Timer3$PT := USINT#0;
            IF Pusher$Timer3$IN THEN
                Pusher$Timer3$Q := (Pusher$Timer3$ET = USINT#0);
                IF (Pusher$Timer3$ET > USINT#0) THEN
                    Pusher$Timer3$ET := (Pusher$Timer3$ET - USINT#1);
                ELSE
                    Pusher$Timer3$ET := USINT#0;
                END_IF;
            ELSE
                Pusher$Timer3$Q := FALSE;
                Pusher$Timer3$ET := Pusher$Timer3$PT;
            END_IF;
            Pusher$interconnect_Slide1_Black := FALSE;
            Pusher$Timer_Slide1_Black$IN := FALSE;
            Pusher$Timer_Slide1_Black$PT := USINT#0;
            IF Pusher$Timer_Slide1_Black$IN THEN
                Pusher$Timer_Slide1_Black$Q := (Pusher$Timer_Slide1_Black$ET = USINT#0);
                IF (Pusher$Timer_Slide1_Black$ET > USINT#0) THEN
                    Pusher$Timer_Slide1_Black$ET := (Pusher$Timer_Slide1_Black$ET - USINT#1);
                ELSE
                    Pusher$Timer_Slide1_Black$ET := USINT#0;
                END_IF;
            ELSE
                Pusher$Timer_Slide1_Black$Q := FALSE;
                Pusher$Timer_Slide1_Black$ET := Pusher$Timer_Slide1_Black$PT;
            END_IF;
            Pusher$Slide1_black := (Pusher$Slide1_black - INT#1);
            Pusher$Priority_Var_Black := (Pusher$Priority_Var_Black - INT#1);
            {* end(onActive) *}
            {* begin(transition) *}
            IF TRUE THEN
                Pusher$_transit := TRUE;
                Pusher$_state := Pusher_states_t#Interstep_2;
            END_IF;
            {* end(transition) *}
            {* begin(onExit) *}
            {* end(onExit) *}
            {* end(State) *}

        Pusher_states_t#Reset_interconnect_Slide1_Metal:
            {* begin(State) *}
            {* begin(onEntry) *}
            Pusher$_transit := FALSE;
            {* end(onEntry) *}
            {* begin(onActive) *}
            Pusher$interconnect3 := FALSE;
            Pusher$Timer3$IN := FALSE;
            Pusher$Timer3$PT := USINT#0;
            IF Pusher$Timer3$IN THEN
                Pusher$Timer3$Q := (Pusher$Timer3$ET = USINT#0);
                IF (Pusher$Timer3$ET > USINT#0) THEN
                    Pusher$Timer3$ET := (Pusher$Timer3$ET - USINT#1);
                ELSE
                    Pusher$Timer3$ET := USINT#0;
                END_IF;
            ELSE
                Pusher$Timer3$Q := FALSE;
                Pusher$Timer3$ET := Pusher$Timer3$PT;
            END_IF;
            Pusher$interconnect_Slide1_Metal := FALSE;
            Pusher$Timer_Slide1_Metal$IN := FALSE;
            Pusher$Timer_Slide1_Metal$PT := USINT#0;
            IF Pusher$Timer_Slide1_Metal$IN THEN
                Pusher$Timer_Slide1_Metal$Q := (Pusher$Timer_Slide1_Metal$ET = USINT#0);
                IF (Pusher$Timer_Slide1_Metal$ET > USINT#0) THEN
                    Pusher$Timer_Slide1_Metal$ET := (Pusher$Timer_Slide1_Metal$ET - USINT#1);
                ELSE
                    Pusher$Timer_Slide1_Metal$ET := USINT#0;
                END_IF;
            ELSE
                Pusher$Timer_Slide1_Metal$Q := FALSE;
                Pusher$Timer_Slide1_Metal$ET := Pusher$Timer_Slide1_Metal$PT;
            END_IF;
            Pusher$Slide1_metal := (Pusher$Slide1_metal - INT#1);
            Pusher$Priority_Var_Metal := (Pusher$Priority_Var_Metal - INT#1);
            {* end(onActive) *}
            {* begin(transition) *}
            IF TRUE THEN
                Pusher$_transit := TRUE;
                Pusher$_state := Pusher_states_t#Interstep_2;
            END_IF;
            {* end(transition) *}
            {* begin(onExit) *}
            {* end(onExit) *}
            {* end(State) *}

        Pusher_states_t#Reset_interconnect_Slide1_White:
            {* begin(State) *}
            {* begin(onEntry) *}
            Pusher$_transit := FALSE;
            {* end(onEntry) *}
            {* begin(onActive) *}
            Pusher$interconnect3 := FALSE;
            Pusher$Timer3$IN := FALSE;
            Pusher$Timer3$PT := USINT#0;
            IF Pusher$Timer3$IN THEN
                Pusher$Timer3$Q := (Pusher$Timer3$ET = USINT#0);
                IF (Pusher$Timer3$ET > USINT#0) THEN
                    Pusher$Timer3$ET := (Pusher$Timer3$ET - USINT#1);
                ELSE
                    Pusher$Timer3$ET := USINT#0;
                END_IF;
            ELSE
                Pusher$Timer3$Q := FALSE;
                Pusher$Timer3$ET := Pusher$Timer3$PT;
            END_IF;
            Pusher$interconnect_Slide1_White := FALSE;
            Pusher$Timer_Slide1_White$IN := FALSE;
            Pusher$Timer_Slide1_White$PT := USINT#0;
            IF Pusher$Timer_Slide1_White$IN THEN
                Pusher$Timer_Slide1_White$Q := (Pusher$Timer_Slide1_White$ET = USINT#0);
                IF (Pusher$Timer_Slide1_White$ET > USINT#0) THEN
                    Pusher$Timer_Slide1_White$ET := (Pusher$Timer_Slide1_White$ET - USINT#1);
                ELSE
                    Pusher$Timer_Slide1_White$ET := USINT#0;
                END_IF;
            ELSE
                Pusher$Timer_Slide1_White$Q := FALSE;
                Pusher$Timer_Slide1_White$ET := Pusher$Timer_Slide1_White$PT;
            END_IF;
            Pusher$Slide1_white := (Pusher$Slide1_white - INT#1);
            Pusher$Priority_Var_White := (Pusher$Priority_Var_White - INT#1);
            {* end(onActive) *}
            {* begin(transition) *}
            IF TRUE THEN
                Pusher$_transit := TRUE;
                Pusher$_state := Pusher_states_t#Interstep_2;
            END_IF;
            {* end(transition) *}
            {* begin(onExit) *}
            {* end(onExit) *}
            {* end(State) *}

        Pusher_states_t#Reset_interconnect_Slide2_Black:
            {* begin(State) *}
            {* begin(onEntry) *}
            Pusher$_transit := FALSE;
            {* end(onEntry) *}
            {* begin(onActive) *}
            Pusher$interconnect3 := FALSE;
            Pusher$Timer3$IN := FALSE;
            Pusher$Timer3$PT := USINT#0;
            IF Pusher$Timer3$IN THEN
                Pusher$Timer3$Q := (Pusher$Timer3$ET = USINT#0);
                IF (Pusher$Timer3$ET > USINT#0) THEN
                    Pusher$Timer3$ET := (Pusher$Timer3$ET - USINT#1);
                ELSE
                    Pusher$Timer3$ET := USINT#0;
                END_IF;
            ELSE
                Pusher$Timer3$Q := FALSE;
                Pusher$Timer3$ET := Pusher$Timer3$PT;
            END_IF;
            Pusher$interconnect_Slide2_Black := FALSE;
            Pusher$Timer_Slide2_Black$IN := FALSE;
            Pusher$Timer_Slide2_Black$PT := USINT#0;
            IF Pusher$Timer_Slide2_Black$IN THEN
                Pusher$Timer_Slide2_Black$Q := (Pusher$Timer_Slide2_Black$ET = USINT#0);
                IF (Pusher$Timer_Slide2_Black$ET > USINT#0) THEN
                    Pusher$Timer_Slide2_Black$ET := (Pusher$Timer_Slide2_Black$ET - USINT#1);
                ELSE
                    Pusher$Timer_Slide2_Black$ET := USINT#0;
                END_IF;
            ELSE
                Pusher$Timer_Slide2_Black$Q := FALSE;
                Pusher$Timer_Slide2_Black$ET := Pusher$Timer_Slide2_Black$PT;
            END_IF;
            Pusher$Slide2_black := (Pusher$Slide2_black - INT#1);
            Pusher$Priority_Var_Black := (Pusher$Priority_Var_Black - INT#1);
            {* end(onActive) *}
            {* begin(transition) *}
            IF TRUE THEN
                Pusher$_transit := TRUE;
                Pusher$_state := Pusher_states_t#Interstep_2;
            END_IF;
            {* end(transition) *}
            {* begin(onExit) *}
            {* end(onExit) *}
            {* end(State) *}

        Pusher_states_t#Reset_interconnect_Slide2_Metal:
            {* begin(State) *}
            {* begin(onEntry) *}
            Pusher$_transit := FALSE;
            {* end(onEntry) *}
            {* begin(onActive) *}
            Pusher$interconnect3 := FALSE;
            Pusher$Timer3$IN := FALSE;
            Pusher$Timer3$PT := USINT#0;
            IF Pusher$Timer3$IN THEN
                Pusher$Timer3$Q := (Pusher$Timer3$ET = USINT#0);
                IF (Pusher$Timer3$ET > USINT#0) THEN
                    Pusher$Timer3$ET := (Pusher$Timer3$ET - USINT#1);
                ELSE
                    Pusher$Timer3$ET := USINT#0;
                END_IF;
            ELSE
                Pusher$Timer3$Q := FALSE;
                Pusher$Timer3$ET := Pusher$Timer3$PT;
            END_IF;
            Pusher$interconnect_Slide2_Metal := FALSE;
            Pusher$Timer_Slide2_Metal$IN := FALSE;
            Pusher$Timer_Slide2_Metal$PT := USINT#0;
            IF Pusher$Timer_Slide2_Metal$IN THEN
                Pusher$Timer_Slide2_Metal$Q := (Pusher$Timer_Slide2_Metal$ET = USINT#0);
                IF (Pusher$Timer_Slide2_Metal$ET > USINT#0) THEN
                    Pusher$Timer_Slide2_Metal$ET := (Pusher$Timer_Slide2_Metal$ET - USINT#1);
                ELSE
                    Pusher$Timer_Slide2_Metal$ET := USINT#0;
                END_IF;
            ELSE
                Pusher$Timer_Slide2_Metal$Q := FALSE;
                Pusher$Timer_Slide2_Metal$ET := Pusher$Timer_Slide2_Metal$PT;
            END_IF;
            Pusher$Slide2_metal := (Pusher$Slide2_metal - INT#1);
            Pusher$Priority_Var_Metal := (Pusher$Priority_Var_Metal - INT#1);
            {* end(onActive) *}
            {* begin(transition) *}
            IF TRUE THEN
                Pusher$_transit := TRUE;
                Pusher$_state := Pusher_states_t#Interstep_2;
            END_IF;
            {* end(transition) *}
            {* begin(onExit) *}
            {* end(onExit) *}
            {* end(State) *}

        Pusher_states_t#Reset_interconnect_Slide2_White:
            {* begin(State) *}
            {* begin(onEntry) *}
            Pusher$_transit := FALSE;
            {* end(onEntry) *}
            {* begin(onActive) *}
            Pusher$interconnect3 := FALSE;
            Pusher$Timer3$IN := FALSE;
            Pusher$Timer3$PT := USINT#0;
            IF Pusher$Timer3$IN THEN
                Pusher$Timer3$Q := (Pusher$Timer3$ET = USINT#0);
                IF (Pusher$Timer3$ET > USINT#0) THEN
                    Pusher$Timer3$ET := (Pusher$Timer3$ET - USINT#1);
                ELSE
                    Pusher$Timer3$ET := USINT#0;
                END_IF;
            ELSE
                Pusher$Timer3$Q := FALSE;
                Pusher$Timer3$ET := Pusher$Timer3$PT;
            END_IF;
            Pusher$interconnect_Slide2_White := FALSE;
            Pusher$Timer_Slide2_White$IN := FALSE;
            Pusher$Timer_Slide2_White$PT := USINT#0;
            IF Pusher$Timer_Slide2_White$IN THEN
                Pusher$Timer_Slide2_White$Q := (Pusher$Timer_Slide2_White$ET = USINT#0);
                IF (Pusher$Timer_Slide2_White$ET > USINT#0) THEN
                    Pusher$Timer_Slide2_White$ET := (Pusher$Timer_Slide2_White$ET - USINT#1);
                ELSE
                    Pusher$Timer_Slide2_White$ET := USINT#0;
                END_IF;
            ELSE
                Pusher$Timer_Slide2_White$Q := FALSE;
                Pusher$Timer_Slide2_White$ET := Pusher$Timer_Slide2_White$PT;
            END_IF;
            Pusher$Slide2_white := (Pusher$Slide2_white - INT#1);
            Pusher$Priority_Var_White := (Pusher$Priority_Var_White - INT#1);
            {* end(onActive) *}
            {* begin(transition) *}
            IF TRUE THEN
                Pusher$_transit := TRUE;
                Pusher$_state := Pusher_states_t#Interstep_2;
            END_IF;
            {* end(transition) *}
            {* begin(onExit) *}
            {* end(onExit) *}
            {* end(State) *}

        Pusher_states_t#Reset_interconnect_Slide3_Metal:
            {* begin(State) *}
            {* begin(onEntry) *}
            Pusher$_transit := FALSE;
            {* end(onEntry) *}
            {* begin(onActive) *}
            Pusher$interconnect3 := FALSE;
            Pusher$Timer3$IN := FALSE;
            Pusher$Timer3$PT := USINT#0;
            IF Pusher$Timer3$IN THEN
                Pusher$Timer3$Q := (Pusher$Timer3$ET = USINT#0);
                IF (Pusher$Timer3$ET > USINT#0) THEN
                    Pusher$Timer3$ET := (Pusher$Timer3$ET - USINT#1);
                ELSE
                    Pusher$Timer3$ET := USINT#0;
                END_IF;
            ELSE
                Pusher$Timer3$Q := FALSE;
                Pusher$Timer3$ET := Pusher$Timer3$PT;
            END_IF;
            Pusher$Slide3_metal := (Pusher$Slide3_metal - INT#1);
            Pusher$Priority_Var_Metal := (Pusher$Priority_Var_Metal - INT#1);
            {* end(onActive) *}
            {* begin(transition) *}
            IF TRUE THEN
                Pusher$_transit := TRUE;
                Pusher$_state := Pusher_states_t#Interstep_2;
            END_IF;
            {* end(transition) *}
            {* begin(onExit) *}
            {* end(onExit) *}
            {* end(State) *}

        Pusher_states_t#Reset_interconnect_Slide3_White:
            {* begin(State) *}
            {* begin(onEntry) *}
            Pusher$_transit := FALSE;
            {* end(onEntry) *}
            {* begin(onActive) *}
            Pusher$interconnect3 := FALSE;
            Pusher$Timer3$IN := FALSE;
            Pusher$Timer3$PT := USINT#0;
            IF Pusher$Timer3$IN THEN
                Pusher$Timer3$Q := (Pusher$Timer3$ET = USINT#0);
                IF (Pusher$Timer3$ET > USINT#0) THEN
                    Pusher$Timer3$ET := (Pusher$Timer3$ET - USINT#1);
                ELSE
                    Pusher$Timer3$ET := USINT#0;
                END_IF;
            ELSE
                Pusher$Timer3$Q := FALSE;
                Pusher$Timer3$ET := Pusher$Timer3$PT;
            END_IF;
            Pusher$Slide3_white := (Pusher$Slide3_white - INT#1);
            Pusher$Priority_Var_White := (Pusher$Priority_Var_White - INT#1);
            {* end(onActive) *}
            {* begin(transition) *}
            IF TRUE THEN
                Pusher$_transit := TRUE;
                Pusher$_state := Pusher_states_t#Interstep_2;
            END_IF;
            {* end(transition) *}
            {* begin(onExit) *}
            {* end(onExit) *}
            {* end(State) *}

        Pusher_states_t#Second_Slide_Timer_Black:
            {* begin(State) *}
            {* begin(onEntry) *}
            Pusher$_transit := FALSE;
            {* end(onEntry) *}
            {* begin(onActive) *}
            IF (Pusher$SorterLightnesssensorCraneInterfaceInverse = TRUE) THEN
                Pusher$Timer_Slide2_Black$IN := Pusher$SorterLightnesssensorCraneInterfaceInverse;
                Pusher$Timer_Slide2_Black$PT := Pusher$Duration_Slide2_Black;
                IF Pusher$Timer_Slide2_Black$IN THEN
                    Pusher$Timer_Slide2_Black$Q := (Pusher$Timer_Slide2_Black$ET = USINT#0);
                    IF (Pusher$Timer_Slide2_Black$ET > USINT#0) THEN
                        Pusher$Timer_Slide2_Black$ET := (Pusher$Timer_Slide2_Black$ET - USINT#1);
                    ELSE
                        Pusher$Timer_Slide2_Black$ET := USINT#0;
                    END_IF;
                ELSE
                    Pusher$Timer_Slide2_Black$Q := FALSE;
                    Pusher$Timer_Slide2_Black$ET := Pusher$Timer_Slide2_Black$PT;
                END_IF;
                Pusher$interconnect_Slide2_Black := Pusher$Timer_Slide2_Black$Q;
            END_IF;
            {* end(onActive) *}
            {* begin(transition) *}
            IF Pusher$interconnect_Slide2_Black THEN
                Pusher$_transit := TRUE;
                Pusher$_state := Pusher_states_t#PusherY2_Move_Out_Black;
            END_IF;
            {* end(transition) *}
            {* begin(onExit) *}
            {* end(onExit) *}
            {* end(State) *}

        Pusher_states_t#Second_Slide_Timer_Metal:
            {* begin(State) *}
            {* begin(onEntry) *}
            Pusher$_transit := FALSE;
            {* end(onEntry) *}
            {* begin(onActive) *}
            Pusher$Timer_Slide2_Metal$IN := TRUE;
            Pusher$Timer_Slide2_Metal$PT := Pusher$Duration_Slide2_Metal;
            IF Pusher$Timer_Slide2_Metal$IN THEN
                Pusher$Timer_Slide2_Metal$Q := (Pusher$Timer_Slide2_Metal$ET = USINT#0);
                IF (Pusher$Timer_Slide2_Metal$ET > USINT#0) THEN
                    Pusher$Timer_Slide2_Metal$ET := (Pusher$Timer_Slide2_Metal$ET - USINT#1);
                ELSE
                    Pusher$Timer_Slide2_Metal$ET := USINT#0;
                END_IF;
            ELSE
                Pusher$Timer_Slide2_Metal$Q := FALSE;
                Pusher$Timer_Slide2_Metal$ET := Pusher$Timer_Slide2_Metal$PT;
            END_IF;
            Pusher$interconnect_Slide2_Metal := Pusher$Timer_Slide2_Metal$Q;
            {* end(onActive) *}
            {* begin(transition) *}
            IF Pusher$interconnect_Slide2_Metal THEN
                Pusher$_transit := TRUE;
                Pusher$_state := Pusher_states_t#PusherY2_Move_Out_Metal;
            END_IF;
            {* end(transition) *}
            {* begin(onExit) *}
            {* end(onExit) *}
            {* end(State) *}

        Pusher_states_t#Second_Slide_Timer_White:
            {* begin(State) *}
            {* begin(onEntry) *}
            Pusher$_transit := FALSE;
            {* end(onEntry) *}
            {* begin(onActive) *}
            Pusher$Timer_Slide2_White$IN := TRUE;
            Pusher$Timer_Slide2_White$PT := Pusher$Duration_Slide2_White;
            IF Pusher$Timer_Slide2_White$IN THEN
                Pusher$Timer_Slide2_White$Q := (Pusher$Timer_Slide2_White$ET = USINT#0);
                IF (Pusher$Timer_Slide2_White$ET > USINT#0) THEN
                    Pusher$Timer_Slide2_White$ET := (Pusher$Timer_Slide2_White$ET - USINT#1);
                ELSE
                    Pusher$Timer_Slide2_White$ET := USINT#0;
                END_IF;
            ELSE
                Pusher$Timer_Slide2_White$Q := FALSE;
                Pusher$Timer_Slide2_White$ET := Pusher$Timer_Slide2_White$PT;
            END_IF;
            Pusher$interconnect_Slide2_White := Pusher$Timer_Slide2_White$Q;
            {* end(onActive) *}
            {* begin(transition) *}
            IF Pusher$interconnect_Slide2_White THEN
                Pusher$_transit := TRUE;
                Pusher$_state := Pusher_states_t#PusherY2_Move_Out_White;
            END_IF;
            {* end(transition) *}
            {* begin(onExit) *}
            {* end(onExit) *}
            {* end(State) *}

        Pusher_states_t#Second_Slide_black_workpieces:
            {* begin(State) *}
            {* begin(onEntry) *}
            Pusher$_transit := FALSE;
            {* end(onEntry) *}
            {* begin(onActive) *}
            {* end(onActive) *}
            {* begin(transition) *}
            IF TRUE THEN
                Pusher$_transit := TRUE;
                Pusher$_state := Pusher_states_t#Second_Slide_Timer_Black;
            END_IF;
            {* end(transition) *}
            {* begin(onExit) *}
            {* end(onExit) *}
            {* end(State) *}

        Pusher_states_t#Second_Slide_metal_workpieces:
            {* begin(State) *}
            {* begin(onEntry) *}
            Pusher$_transit := FALSE;
            {* end(onEntry) *}
            {* begin(onActive) *}
            {* end(onActive) *}
            {* begin(transition) *}
            IF (Pusher$SorterLightnessSensorPusher2 AND Pusher$SorterCapacitiveSensorPusher2) THEN
                Pusher$_transit := TRUE;
                Pusher$_state := Pusher_states_t#Second_Test_For_Metal;
            END_IF;
            {* end(transition) *}
            {* begin(onExit) *}
            {* end(onExit) *}
            {* end(State) *}

        Pusher_states_t#Second_Slide_white_workpieces:
            {* begin(State) *}
            {* begin(onEntry) *}
            Pusher$_transit := FALSE;
            {* end(onEntry) *}
            {* begin(onActive) *}
            {* end(onActive) *}
            {* begin(transition) *}
            IF (Pusher$SorterLightnessSensorPusher2 AND NOT Pusher$SorterCapacitiveSensorPusher2) THEN
                Pusher$_transit := TRUE;
                Pusher$_state := Pusher_states_t#Second_Test_For_White;
            END_IF;
            {* end(transition) *}
            {* begin(onExit) *}
            {* end(onExit) *}
            {* end(State) *}

        Pusher_states_t#Second_Test_For_Metal:
            {* begin(State) *}
            {* begin(onEntry) *}
            Pusher$_transit := FALSE;
            {* end(onEntry) *}
            {* begin(onActive) *}
            {* end(onActive) *}
            {* begin(transition) *}
            IF TRUE THEN
                Pusher$_transit := TRUE;
                Pusher$_state := Pusher_states_t#Second_Slide_Timer_Metal;
            END_IF;
            {* end(transition) *}
            {* begin(onExit) *}
            {* end(onExit) *}
            {* end(State) *}

        Pusher_states_t#Second_Test_For_White:
            {* begin(State) *}
            {* begin(onEntry) *}
            Pusher$_transit := FALSE;
            {* end(onEntry) *}
            {* begin(onActive) *}
            {* end(onActive) *}
            {* begin(transition) *}
            IF TRUE THEN
                Pusher$_transit := TRUE;
                Pusher$_state := Pusher_states_t#Second_Slide_Timer_White;
            END_IF;
            {* end(transition) *}
            {* begin(onExit) *}
            {* end(onExit) *}
            {* end(State) *}

        Pusher_states_t#Third_Slide_black_workpieces:
            {* begin(State) *}
            {* begin(onEntry) *}
            Pusher$_transit := FALSE;
            {* end(onEntry) *}
            {* begin(onActive) *}
            {* end(onActive) *}
            {* begin(transition) *}
            IF (NOT Pusher$SorterLightnessSensorPusher2 AND NOT Pusher$SorterCapacitiveSensorPusher2) THEN
                Pusher$_transit := TRUE;
                Pusher$_state := Pusher_states_t#Wait_Black;
            END_IF;
            {* end(transition) *}
            {* begin(onExit) *}
            {* end(onExit) *}
            {* end(State) *}

        Pusher_states_t#Third_Slide_metal_workpieces:
            {* begin(State) *}
            {* begin(onEntry) *}
            Pusher$_transit := FALSE;
            {* end(onEntry) *}
            {* begin(onActive) *}
            {* end(onActive) *}
            {* begin(transition) *}
            IF (Pusher$SorterLightnessSensorPusher2 AND Pusher$SorterCapacitiveSensorPusher2) THEN
                Pusher$_transit := TRUE;
                Pusher$_state := Pusher_states_t#Wait_Metal;
            END_IF;
            {* end(transition) *}
            {* begin(onExit) *}
            {* end(onExit) *}
            {* end(State) *}

        Pusher_states_t#Third_Slide_white_workpieces:
            {* begin(State) *}
            {* begin(onEntry) *}
            Pusher$_transit := FALSE;
            {* end(onEntry) *}
            {* begin(onActive) *}
            {* end(onActive) *}
            {* begin(transition) *}
            IF (Pusher$SorterLightnessSensorPusher2 AND NOT Pusher$SorterCapacitiveSensorPusher2) THEN
                Pusher$_transit := TRUE;
                Pusher$_state := Pusher_states_t#Wait_White;
            END_IF;
            {* end(transition) *}
            {* begin(onExit) *}
            {* end(onExit) *}
            {* end(State) *}

        Pusher_states_t#Wait_Black:
            {* begin(State) *}
            {* begin(onEntry) *}
            Pusher$_transit := FALSE;
            {* end(onEntry) *}
            {* begin(onActive) *}
            IF ((NOT Pusher$SorterLightnessSensorPusher2 AND NOT Pusher$SorterCapacitiveSensorPusher2) = TRUE) THEN
                Pusher$Timer2$IN := (NOT Pusher$SorterLightnessSensorPusher2 AND NOT Pusher$SorterCapacitiveSensorPusher2);
                Pusher$Timer2$PT := Pusher$Duration2;
                IF Pusher$Timer2$IN THEN
                    Pusher$Timer2$Q := (Pusher$Timer2$ET = USINT#0);
                    IF (Pusher$Timer2$ET > USINT#0) THEN
                        Pusher$Timer2$ET := (Pusher$Timer2$ET - USINT#1);
                    ELSE
                        Pusher$Timer2$ET := USINT#0;
                    END_IF;
                ELSE
                    Pusher$Timer2$Q := FALSE;
                    Pusher$Timer2$ET := Pusher$Timer2$PT;
                END_IF;
                Pusher$interconnect2 := Pusher$Timer2$Q;
            END_IF;
            {* end(onActive) *}
            {* begin(transition) *}
            IF Pusher$interconnect2 THEN
                Pusher$_transit := TRUE;
                Pusher$_state := Pusher_states_t#Reset_interconnect3;
            END_IF;
            {* end(transition) *}
            {* begin(onExit) *}
            {* end(onExit) *}
            {* end(State) *}

        Pusher_states_t#Wait_Metal:
            {* begin(State) *}
            {* begin(onEntry) *}
            Pusher$_transit := FALSE;
            {* end(onEntry) *}
            {* begin(onActive) *}
            Pusher$Timer3$IN := TRUE;
            Pusher$Timer3$PT := Pusher$Duration3;
            IF Pusher$Timer3$IN THEN
                Pusher$Timer3$Q := (Pusher$Timer3$ET = USINT#0);
                IF (Pusher$Timer3$ET > USINT#0) THEN
                    Pusher$Timer3$ET := (Pusher$Timer3$ET - USINT#1);
                ELSE
                    Pusher$Timer3$ET := USINT#0;
                END_IF;
            ELSE
                Pusher$Timer3$Q := FALSE;
                Pusher$Timer3$ET := Pusher$Timer3$PT;
            END_IF;
            Pusher$interconnect3 := Pusher$Timer3$Q;
            {* end(onActive) *}
            {* begin(transition) *}
            IF Pusher$interconnect3 THEN
                Pusher$_transit := TRUE;
                Pusher$_state := Pusher_states_t#Reset_interconnect_Slide3_Metal;
            END_IF;
            {* end(transition) *}
            {* begin(onExit) *}
            {* end(onExit) *}
            {* end(State) *}

        Pusher_states_t#Wait_White:
            {* begin(State) *}
            {* begin(onEntry) *}
            Pusher$_transit := FALSE;
            {* end(onEntry) *}
            {* begin(onActive) *}
            Pusher$Timer3$IN := TRUE;
            Pusher$Timer3$PT := Pusher$Duration3;
            IF Pusher$Timer3$IN THEN
                Pusher$Timer3$Q := (Pusher$Timer3$ET = USINT#0);
                IF (Pusher$Timer3$ET > USINT#0) THEN
                    Pusher$Timer3$ET := (Pusher$Timer3$ET - USINT#1);
                ELSE
                    Pusher$Timer3$ET := USINT#0;
                END_IF;
            ELSE
                Pusher$Timer3$Q := FALSE;
                Pusher$Timer3$ET := Pusher$Timer3$PT;
            END_IF;
            Pusher$interconnect3 := Pusher$Timer3$Q;
            {* end(onActive) *}
            {* begin(transition) *}
            IF Pusher$interconnect3 THEN
                Pusher$_transit := TRUE;
                Pusher$_state := Pusher_states_t#Reset_interconnect_Slide3_White;
            END_IF;
            {* end(transition) *}
            {* begin(onExit) *}
            {* end(onExit) *}
            {* end(State) *}

        Pusher_states_t#Wait_Y1_Black:
            {* begin(State) *}
            {* begin(onEntry) *}
            Pusher$_transit := FALSE;
            {* end(onEntry) *}
            {* begin(onActive) *}
            IF (Pusher$PusherY1 = TRUE) THEN
                Pusher$Timer3$IN := Pusher$PusherY1;
                Pusher$Timer3$PT := Pusher$Duration3;
                IF Pusher$Timer3$IN THEN
                    Pusher$Timer3$Q := (Pusher$Timer3$ET = USINT#0);
                    IF (Pusher$Timer3$ET > USINT#0) THEN
                        Pusher$Timer3$ET := (Pusher$Timer3$ET - USINT#1);
                    ELSE
                        Pusher$Timer3$ET := USINT#0;
                    END_IF;
                ELSE
                    Pusher$Timer3$Q := FALSE;
                    Pusher$Timer3$ET := Pusher$Timer3$PT;
                END_IF;
                Pusher$interconnect3 := Pusher$Timer3$Q;
            END_IF;
            {* end(onActive) *}
            {* begin(transition) *}
            IF Pusher$interconnect3 THEN
                Pusher$_transit := TRUE;
                Pusher$_state := Pusher_states_t#PusherY1_Move_In_Black;
            END_IF;
            {* end(transition) *}
            {* begin(onExit) *}
            {* end(onExit) *}
            {* end(State) *}

        Pusher_states_t#Wait_Y1_Metal:
            {* begin(State) *}
            {* begin(onEntry) *}
            Pusher$_transit := FALSE;
            {* end(onEntry) *}
            {* begin(onActive) *}
            IF (Pusher$PusherY1 = TRUE) THEN
                Pusher$Timer3$IN := Pusher$PusherY1;
                Pusher$Timer3$PT := Pusher$Duration3;
                IF Pusher$Timer3$IN THEN
                    Pusher$Timer3$Q := (Pusher$Timer3$ET = USINT#0);
                    IF (Pusher$Timer3$ET > USINT#0) THEN
                        Pusher$Timer3$ET := (Pusher$Timer3$ET - USINT#1);
                    ELSE
                        Pusher$Timer3$ET := USINT#0;
                    END_IF;
                ELSE
                    Pusher$Timer3$Q := FALSE;
                    Pusher$Timer3$ET := Pusher$Timer3$PT;
                END_IF;
                Pusher$interconnect3 := Pusher$Timer3$Q;
            END_IF;
            {* end(onActive) *}
            {* begin(transition) *}
            IF Pusher$interconnect3 THEN
                Pusher$_transit := TRUE;
                Pusher$_state := Pusher_states_t#PusherY1_Move_In_Metal;
            END_IF;
            {* end(transition) *}
            {* begin(onExit) *}
            {* end(onExit) *}
            {* end(State) *}

        Pusher_states_t#Wait_Y1_White:
            {* begin(State) *}
            {* begin(onEntry) *}
            Pusher$_transit := FALSE;
            {* end(onEntry) *}
            {* begin(onActive) *}
            IF (Pusher$PusherY1 = TRUE) THEN
                Pusher$Timer3$IN := Pusher$PusherY1;
                Pusher$Timer3$PT := Pusher$Duration3;
                IF Pusher$Timer3$IN THEN
                    Pusher$Timer3$Q := (Pusher$Timer3$ET = USINT#0);
                    IF (Pusher$Timer3$ET > USINT#0) THEN
                        Pusher$Timer3$ET := (Pusher$Timer3$ET - USINT#1);
                    ELSE
                        Pusher$Timer3$ET := USINT#0;
                    END_IF;
                ELSE
                    Pusher$Timer3$Q := FALSE;
                    Pusher$Timer3$ET := Pusher$Timer3$PT;
                END_IF;
                Pusher$interconnect3 := Pusher$Timer3$Q;
            END_IF;
            {* end(onActive) *}
            {* begin(transition) *}
            IF Pusher$interconnect3 THEN
                Pusher$_transit := TRUE;
                Pusher$_state := Pusher_states_t#PusherY1_Move_In_White;
            END_IF;
            {* end(transition) *}
            {* begin(onExit) *}
            {* end(onExit) *}
            {* end(State) *}

        Pusher_states_t#Wait_Y2_Black:
            {* begin(State) *}
            {* begin(onEntry) *}
            Pusher$_transit := FALSE;
            {* end(onEntry) *}
            {* begin(onActive) *}
            IF (Pusher$PusherY2 = TRUE) THEN
                Pusher$Timer3$IN := Pusher$PusherY2;
                Pusher$Timer3$PT := Pusher$Duration3;
                IF Pusher$Timer3$IN THEN
                    Pusher$Timer3$Q := (Pusher$Timer3$ET = USINT#0);
                    IF (Pusher$Timer3$ET > USINT#0) THEN
                        Pusher$Timer3$ET := (Pusher$Timer3$ET - USINT#1);
                    ELSE
                        Pusher$Timer3$ET := USINT#0;
                    END_IF;
                ELSE
                    Pusher$Timer3$Q := FALSE;
                    Pusher$Timer3$ET := Pusher$Timer3$PT;
                END_IF;
                Pusher$interconnect3 := Pusher$Timer3$Q;
            END_IF;
            {* end(onActive) *}
            {* begin(transition) *}
            IF Pusher$interconnect3 THEN
                Pusher$_transit := TRUE;
                Pusher$_state := Pusher_states_t#PusherY2_Move_In_Black;
            END_IF;
            {* end(transition) *}
            {* begin(onExit) *}
            {* end(onExit) *}
            {* end(State) *}

        Pusher_states_t#Wait_Y2_Metal:
            {* begin(State) *}
            {* begin(onEntry) *}
            Pusher$_transit := FALSE;
            {* end(onEntry) *}
            {* begin(onActive) *}
            IF (Pusher$PusherY2 = TRUE) THEN
                Pusher$Timer3$IN := Pusher$PusherY2;
                Pusher$Timer3$PT := Pusher$Duration3;
                IF Pusher$Timer3$IN THEN
                    Pusher$Timer3$Q := (Pusher$Timer3$ET = USINT#0);
                    IF (Pusher$Timer3$ET > USINT#0) THEN
                        Pusher$Timer3$ET := (Pusher$Timer3$ET - USINT#1);
                    ELSE
                        Pusher$Timer3$ET := USINT#0;
                    END_IF;
                ELSE
                    Pusher$Timer3$Q := FALSE;
                    Pusher$Timer3$ET := Pusher$Timer3$PT;
                END_IF;
                Pusher$interconnect3 := Pusher$Timer3$Q;
            END_IF;
            {* end(onActive) *}
            {* begin(transition) *}
            IF Pusher$interconnect3 THEN
                Pusher$_transit := TRUE;
                Pusher$_state := Pusher_states_t#PusherY2_Move_In_Metal;
            END_IF;
            {* end(transition) *}
            {* begin(onExit) *}
            {* end(onExit) *}
            {* end(State) *}

        Pusher_states_t#Wait_Y2_White:
            {* begin(State) *}
            {* begin(onEntry) *}
            Pusher$_transit := FALSE;
            {* end(onEntry) *}
            {* begin(onActive) *}
            IF (Pusher$PusherY2 = TRUE) THEN
                Pusher$Timer3$IN := Pusher$PusherY2;
                Pusher$Timer3$PT := Pusher$Duration3;
                IF Pusher$Timer3$IN THEN
                    Pusher$Timer3$Q := (Pusher$Timer3$ET = USINT#0);
                    IF (Pusher$Timer3$ET > USINT#0) THEN
                        Pusher$Timer3$ET := (Pusher$Timer3$ET - USINT#1);
                    ELSE
                        Pusher$Timer3$ET := USINT#0;
                    END_IF;
                ELSE
                    Pusher$Timer3$Q := FALSE;
                    Pusher$Timer3$ET := Pusher$Timer3$PT;
                END_IF;
                Pusher$interconnect3 := Pusher$Timer3$Q;
            END_IF;
            {* end(onActive) *}
            {* begin(transition) *}
            IF Pusher$interconnect3 THEN
                Pusher$_transit := TRUE;
                Pusher$_state := Pusher_states_t#PusherY2_Move_In_White;
            END_IF;
            {* end(transition) *}
            {* begin(onExit) *}
            {* end(onExit) *}
            {* end(State) *}

            END_CASE;
    IF ((Actuator_SorterGreenLampConveyor AND Actuator_MagazinGreenLamp) AND Actuator_StampGreenLamp) THEN
        IF (((Stamp$StartCommandStamp AND Crane$StartCommandCrane) AND Conveyor$StartCommandConveyor) AND Mag$StartCommandMagazin) THEN
            Crane$StartVar := TRUE;
            Conveyor$StartVar := TRUE;
            Mag$StartVar := TRUE;
            Pusher$StartVar := TRUE;
            Stamp$StartVar := TRUE;
        END_IF;
    END_IF;
    Crane$SFCReset := FALSE;
    Conveyor$SFCReset := FALSE;
    Mag$SFCReset := FALSE;
    Pusher$SFCReset := FALSE;
    Stamp$SFCReset := FALSE;
ELSEIF ((NOT Sensor_SorterEmergencyStop OR NOT Sensor_StampEmergencyStop) OR NOT Sensor_MagazinEmergencyStop) THEN
    Actuator_MagazinSlider := FALSE;
    Actuator_CraneLower := FALSE;
    Actuator_MagazinVacuumOn := FALSE;
    Actuator_MagazinVacuumOff := TRUE;
    Actuator_MagazinGreenLamp := FALSE;
    Actuator_CraneTurnCounterclockwise := FALSE;
    Actuator_CraneTurnClockwise := FALSE;
    Actuator_SorterConveyorTowardsStacker := FALSE;
    Actuator_SorterConveyorTowardsCrane := FALSE;
    Actuator_SorterGreenLampConveyor := FALSE;
    Actuator_PusherY1 := FALSE;
    Actuator_PusherY2 := FALSE;
    Actuator_StampSliderMovedOut := TRUE;
    Actuator_StampSliderMovedIn := FALSE;
    Actuator_StampGreenLamp := FALSE;
    Actuator_StampPusher := FALSE;
    Actuator_AnalogCranePressure := INT#0;
    Crane$SFCReset := TRUE;
    Conveyor$SFCReset := TRUE;
    Mag$SFCReset := TRUE;
    Pusher$SFCReset := TRUE;
    Stamp$SFCReset := TRUE;
    Crane$StartVar := FALSE;
    Conveyor$StartVar := FALSE;
    Mag$StartVar := FALSE;
    Pusher$StartVar := FALSE;
    Stamp$StartVar := FALSE;
END_IF;
END_PROGRAM

(* ---- Scenario13_Final.xml_Main.st ---- *)
PROGRAM Main

VAR  Actuator_AnalogCranePressure : INT; END_VAR {*Lrwxp*}
VAR  Actuator_CraneLower : BOOL; END_VAR {*Lrwxp*}
VAR  Actuator_CraneTurnClockwise : BOOL; END_VAR {*Lrwxp*}
VAR  Actuator_CraneTurnCounterclockwise : BOOL; END_VAR {*Lrwxp*}
VAR  Actuator_MagazinGreenLamp : BOOL; END_VAR {*Lrwxp*}
VAR  Actuator_MagazinSlider : BOOL; END_VAR {*Lrwxp*}
VAR  Actuator_MagazinVacuumOff : BOOL; END_VAR {*Lrwxp*}
VAR  Actuator_MagazinVacuumOn : BOOL; END_VAR {*Lrwxp*}
VAR  Actuator_MagazinWhiteLamp : BOOL; END_VAR {*Lrwxp*}
VAR  Actuator_PusherY1 : BOOL; END_VAR {*Lrwxp*}
VAR  Actuator_PusherY2 : BOOL; END_VAR {*Lrwxp*}
VAR  Actuator_SorterConveyorTowardsCrane : BOOL; END_VAR {*Lrwxp*}
VAR  Actuator_SorterConveyorTowardsStacker : BOOL; END_VAR {*Lrwxp*}
VAR  Actuator_SorterGreenLampConveyor : BOOL; END_VAR {*Lrwxp*}
VAR  Actuator_SorterWhiteLampConveyor : BOOL; END_VAR {*Lrwxp*}
VAR  Actuator_StampGreenLamp : BOOL; END_VAR {*Lrwxp*}
VAR  Actuator_StampPusher : BOOL; END_VAR {*Lrwxp*}
VAR  Actuator_StampSliderMovedIn : BOOL; END_VAR {*Lrwxp*}
VAR  Actuator_StampSliderMovedOut : BOOL; END_VAR {*Lrwxp*}
VAR  Actuator_StampWhiteLamp : BOOL; END_VAR {*Lrwxp*}
VAR  Conveyor : Conveyor; END_VAR {*Lrwxp*}
VAR  Crane : Crane; END_VAR {*Lrwxp*}
VAR  Mag : Magazin; END_VAR {*Lrwxp*}
VAR  Pusher : Pusher; END_VAR {*Lrwxp*}
VAR  Sensor_AnalogCranePosition : INT; END_VAR {*Lrwxp*}
VAR  Sensor_CraneDown : BOOL; END_VAR {*Lrwxp*}
VAR  Sensor_CraneOnConveyor : BOOL; END_VAR {*Lrwxp*}
VAR  Sensor_CraneOnMagazin : BOOL; END_VAR {*Lrwxp*}
VAR  Sensor_CranePosition : BOOL; END_VAR {*Lrwxp*}
VAR  Sensor_CranePositionStamp : BOOL; END_VAR {*Lrwxp*}
VAR  Sensor_CraneSucked : BOOL; END_VAR {*Lrwxp*}
VAR  Sensor_CraneUp : BOOL; END_VAR {*Lrwxp*}
VAR  Sensor_MagazinCapacitiveSensor : BOOL; END_VAR {*Lrwxp*}
VAR  Sensor_MagazinEmergencyStop : BOOL; END_VAR {*Lrwxp*}
VAR  Sensor_MagazinOpticalSensor : BOOL; END_VAR {*Lrwxp*}
VAR  Sensor_MagazinSwitchManuellAutomatic : BOOL; END_VAR {*Lrwxp*}
VAR  Sensor_SliderMovedOut : BOOL; END_VAR {*Lrwxp*}
VAR  Sensor_SliderNotMovedOut : BOOL; END_VAR {*Lrwxp*}
VAR  Sensor_SorterCapacitiveSensorPusher1 : BOOL; END_VAR {*Lrwxp*}
VAR  Sensor_SorterCapacitiveSensorPusher2 : BOOL; END_VAR {*Lrwxp*}
VAR  Sensor_SorterEmergencyStop : BOOL; END_VAR {*Lrwxp*}
VAR  Sensor_SorterLightbarrierCraneInterface : BOOL; END_VAR {*Lrwxp*}
VAR  Sensor_SorterLightnessSensorPusher1 : BOOL; END_VAR {*Lrwxp*}
VAR  Sensor_SorterLightnessSensorPusher2 : BOOL; END_VAR {*Lrwxp*}
VAR  Sensor_SorterLightnessSensorPusher3 : BOOL; END_VAR {*Lrwxp*}
VAR  Sensor_SorterLightnesssensorCraneInterfaceInverse : BOOL; END_VAR {*Lrwxp*}
VAR  Sensor_SorterPusher1MovedIn : BOOL; END_VAR {*Lrwxp*}
VAR  Sensor_SorterPusher1MovedOut : BOOL; END_VAR {*Lrwxp*}
VAR  Sensor_SorterPusher2MovedIn : BOOL; END_VAR {*Lrwxp*}
VAR  Sensor_SorterPusher2MovedOut : BOOL; END_VAR {*Lrwxp*}
VAR  Sensor_SorterStartButton : BOOL; END_VAR {*Lrwxp*}
VAR  Sensor_SorterSwitchManuellAutomatic : BOOL; END_VAR {*Lrwxp*}
VAR  Sensor_StampEmergencyStop : BOOL; END_VAR {*Lrwxp*}
VAR  Sensor_StampLowered : BOOL; END_VAR {*Lrwxp*}
VAR  Sensor_StampSliderFilled : BOOL; END_VAR {*Lrwxp*}
VAR  Sensor_StampSliderSensorMovedIn : BOOL; END_VAR {*Lrwxp*}
VAR  Sensor_StampSliderSensorMovedOut : BOOL; END_VAR {*Lrwxp*}
VAR  Sensor_StampStartButton : BOOL; END_VAR {*Lrwxp*}
VAR  Sensor_StampSwitchManuellAutomatic : BOOL; END_VAR {*Lrwxp*}
VAR  Sensor_StampUp : BOOL; END_VAR {*Lrwxp*}
VAR  Sensor_StartButtonMagazin : BOOL; END_VAR {*Lrwxp*}
VAR  Sensor_WorkpieceReady : BOOL; END_VAR {*Lrwxp*}
VAR  Stamp : Stamp; END_VAR {*Lrwxp*}
Mag.SliderNotMovedOut := Sensor_SliderNotMovedOut;
Mag.SliderMovedOut := Sensor_SliderMovedOut;
Mag.CraneOnMagazin := Sensor_CraneOnMagazin;
Mag.CraneDown := Sensor_CraneDown;
Mag.CraneUp := Sensor_CraneUp;
Mag.CraneOnConveyor := Sensor_CraneOnConveyor;
Mag.WorkpieceReady := Sensor_WorkpieceReady;
Mag.AnalogCranePosition := Sensor_AnalogCranePosition;
Mag.StartButtonMagazin := Sensor_StartButtonMagazin;
Actuator_MagazinSlider := Mag.MagazinSlider;
Actuator_MagazinGreenLamp := Mag.MagazinGreenLamp;
Crane.CraneUp := Sensor_CraneUp;
Crane.CraneDown := Sensor_CraneDown;
Crane.CraneSucked := Sensor_CraneSucked;
Crane.MagazinCapacitiveSensor := Sensor_MagazinCapacitiveSensor;
Crane.SliderMovedOut := Sensor_SliderMovedOut;
Crane.WorkpieceReady := Sensor_WorkpieceReady;
Crane.MagazinOpticalSensor := Sensor_MagazinOpticalSensor;
Crane.StampSliderFilled := Sensor_StampSliderFilled;
Crane.StampSliderSensorMovedOut := Sensor_StampSliderSensorMovedOut;
Crane.StampLowered := Sensor_StampLowered;
Crane.AnalogCranePosition := Sensor_AnalogCranePosition;
Crane.StartButtonMagazin := Sensor_StartButtonMagazin;
Actuator_CraneTurnCounterclockwise := Crane.CraneTurnCounterclockwise;
Actuator_CraneTurnClockwise := Crane.CraneTurnClockwise;
Actuator_CraneLower := Crane.CraneLower;
Actuator_MagazinVacuumOff := Crane.MagazinVacuumOff;
Actuator_MagazinVacuumOn := Crane.MagazinVacuumOn;
Actuator_AnalogCranePressure := Crane.AnalogCranePressure;
Stamp.StampSliderSensorMovedOut := Sensor_StampSliderSensorMovedOut;
Stamp.StampSliderSensorMovedIn := Sensor_StampSliderSensorMovedIn;
Stamp.StampSliderFilled := Sensor_StampSliderFilled;
Stamp.StampUp := Sensor_StampUp;
Stamp.StampLowered := Sensor_StampLowered;
Stamp.CraneDown := Sensor_CraneDown;
Stamp.CraneUp := Sensor_CraneUp;
Stamp.CraneSucked := Sensor_CraneSucked;
Stamp.CranePositionStamp := Sensor_CranePositionStamp;
Stamp.CraneOnConveyor := Sensor_CraneOnConveyor;
Stamp.AnalogCranePosition := Sensor_AnalogCranePosition;
Stamp.StampStartButton := Sensor_StampStartButton;
Actuator_StampSliderMovedOut := Stamp.StampSliderMovedOut;
Actuator_StampSliderMovedIn := Stamp.StampSliderMovedIn;
Actuator_StampWhiteLamp := Stamp.StampWhiteLamp;
Actuator_StampPusher := Stamp.StampPusher;
Actuator_StampGreenLamp := Stamp.StampGreenLamp;
Conveyor.SorterStartButton := Sensor_SorterStartButton;
Conveyor.SorterSwitchManuellAutomatic := Sensor_SorterSwitchManuellAutomatic;
Conveyor.SorterLightbarrierCraneInterface := Sensor_SorterLightbarrierCraneInterface;
Actuator_SorterConveyorTowardsStacker := Conveyor.SorterConveyorTowardsStacker;
Actuator_SorterConveyorTowardsCrane := Conveyor.SorterConveyorTowardsCrane;
Actuator_SorterGreenLampConveyor := Conveyor.SorterGreenLampConveyor;
Actuator_SorterWhiteLampConveyor := Conveyor.SorterWhiteLampConveyor;
Pusher.SorterLightnesssensorCraneInterfaceInverse := Sensor_SorterLightnesssensorCraneInterfaceInverse;
Pusher.SorterLightbarrierCraneInterface := Sensor_SorterLightbarrierCraneInterface;
Pusher.SorterCapacitiveSensorPusher1 := Sensor_SorterCapacitiveSensorPusher1;
Pusher.SorterLightnessSensorPusher1 := Sensor_SorterLightnessSensorPusher1;
Pusher.SorterCapacitiveSensorPusher2 := Sensor_SorterCapacitiveSensorPusher2;
Pusher.SorterLightnessSensorPusher2 := Sensor_SorterLightnessSensorPusher2;
Pusher.SorterLightnessSensorPusher3 := Sensor_SorterLightnessSensorPusher3;
Pusher.SorterPusher1MovedOut := Sensor_SorterPusher1MovedOut;
Pusher.SorterPusher1MovedIn := Sensor_SorterPusher1MovedIn;
Pusher.SorterPusher2MovedOut := Sensor_SorterPusher2MovedOut;
Pusher.SorterPusher2MovedIn := Sensor_SorterPusher2MovedIn;
Pusher.SorterStartButton := Sensor_SorterStartButton;
Actuator_PusherY1 := Pusher.PusherY1;
Actuator_PusherY2 := Pusher.PusherY2;
IF ((Sensor_SorterEmergencyStop AND Sensor_StampEmergencyStop) AND Sensor_MagazinEmergencyStop) THEN
    Mag();
    Crane();
    Stamp();
    Conveyor();
    Pusher();
    IF ((Actuator_SorterGreenLampConveyor AND Actuator_MagazinGreenLamp) AND Actuator_StampGreenLamp) THEN
        IF (((Stamp.StartCommandStamp AND Crane.StartCommandCrane) AND Conveyor.StartCommandConveyor) AND Mag.StartCommandMagazin) THEN
            Crane.StartVar := TRUE;
            Conveyor.StartVar := TRUE;
            Mag.StartVar := TRUE;
            Pusher.StartVar := TRUE;
            Stamp.StartVar := TRUE;
        END_IF;
    END_IF;
    Crane.SFCReset := FALSE;
    Conveyor.SFCReset := FALSE;
    Mag.SFCReset := FALSE;
    Pusher.SFCReset := FALSE;
    Stamp.SFCReset := FALSE;
ELSEIF ((NOT Sensor_SorterEmergencyStop OR NOT Sensor_StampEmergencyStop) OR NOT Sensor_MagazinEmergencyStop) THEN
    Actuator_MagazinSlider := FALSE;
    Actuator_CraneLower := FALSE;
    Actuator_MagazinVacuumOn := FALSE;
    Actuator_MagazinVacuumOff := TRUE;
    Actuator_MagazinGreenLamp := FALSE;
    Actuator_CraneTurnCounterclockwise := FALSE;
    Actuator_CraneTurnClockwise := FALSE;
    Actuator_SorterConveyorTowardsStacker := FALSE;
    Actuator_SorterConveyorTowardsCrane := FALSE;
    Actuator_SorterGreenLampConveyor := FALSE;
    Actuator_PusherY1 := FALSE;
    Actuator_PusherY2 := FALSE;
    Actuator_StampSliderMovedOut := TRUE;
    Actuator_StampSliderMovedIn := FALSE;
    Actuator_StampGreenLamp := FALSE;
    Actuator_StampPusher := FALSE;
    Actuator_AnalogCranePressure := INT#0;
    Crane.SFCReset := TRUE;
    Conveyor.SFCReset := TRUE;
    Mag.SFCReset := TRUE;
    Pusher.SFCReset := TRUE;
    Stamp.SFCReset := TRUE;
    Crane.StartVar := FALSE;
    Conveyor.StartVar := FALSE;
    Mag.StartVar := FALSE;
    Pusher.StartVar := FALSE;
    Stamp.StartVar := FALSE;
END_IF;
END_PROGRAM
